// TIA Portal project "Bachelor2024" (V14)

(* hardware
DEVICE "S7-1200 station_1"  S7-1200 Station
   slot 0: "Rack_0"  S7-1200 Rack  Rack  V1.0
   slot 1: "PROFIBUS PLC"  CPU 1212C DC/DC/DC  6ES7 212-1AE40-0XB0  V4.1
   slot 101: "CM 1243-5"  CM 1243-5  6GK7 243-5DX30-0XE0  V1.3
DEVICE "GSD device_1"  GSD.Device
   slot 0: "Rack_0"  Rail
DEVICE "GSD device_2"  GSD.Device
   slot 0: "Rack_0"  Rail
DEVICE "S7-1200 station_2"  S7-1200 Station
   slot 0: "Rack_0"  S7-1200 Rack  Rack  V1.0
   slot 1: "PROFINET PLC"  CPU 1211C AC/DC/Rly  6ES7 211-1BE40-0XB0  V4.2
DEVICE "GSD device_3"  GSD.Device.PN
   slot 0: "Rack"  Rack  V1.0
   slot 0: "COUPLER (PN)"  DP/PN Coupler V1  700-158-3DP01  V 1
      slot 0: "DP/PN Coupler V1"  DP/PN Coupler V1
      slot 1: "PN-IO"  PN-IO
         slot 1: "Port 1"  Port 1
         slot 2: "Port 2"  Port 2
   slot 1: "OUT   2 Bytes_1"  OUT   2 Bytes
      slot 0: "OUT   2 Bytes"  OUT   2 Bytes
   slot 2: "IN   2 Bytes_1"  IN   2 Bytes
      slot 0: "IN   2 Bytes"  IN   2 Bytes
DEVICE "HMI"  KTP700 Basic DP
   slot 0: "KTP700 Basic DP"  KTP700 Basic DP  6AV2 123-2GA03-0AX0  14.0.1.0
   slot 1: "HMI_RT_1"  KTP700 Basic DP  6AV2 123-2GA03-0AX0  14.0.1.0
   slot 7: "HMI.MPI/DP_CP_1"  MPI/DP Interface  14.0.1.0
*)

// ===== PLC "PROFIBUS PLC"  CPU 1212C DC/DC/DC =====

VAR_GLOBAL   // PLC tag table "PUSHBUTTONS"
   "PUSHBUTTON_WHITE" AT %I0.0 : Bool;
   "PUSHBUTTON_BLUE" AT %I0.1 : Bool;
   "PUSHBUTTON_GREEN" AT %I0.2 : Bool;
   "PUSHBUTTON_ORANGE1" AT %I0.3 : Bool;
   "PUSHBUTTON_ORANGE2" AT %I0.4 : Bool;
   "PUSHBUTTON_RED" AT %I0.5 : Bool;
END_VAR

VAR_GLOBAL   // PLC tag table "FAULTS"
   "B_BREAK" AT %Q0.0 : Bool;
   "BA_BREAK" AT %Q0.1 : Bool;
   "TERMINATION_OFF" AT %Q0.2 : Bool;
   "BA_SWITCH" AT %Q0.3 : Bool;
   "NO_GROUNDING" AT %Q0.4 : Bool;
   "BA_SHORT" AT %Q0.5 : Bool;
END_VAR

VAR_GLOBAL   // PLC tag table "TESTBOARD_COUPLER"
   "TESTBOARD_INPUT1" AT %IB1 : Byte;
   "TESTBOARD_INPUT2" AT %IB2 : Byte;
   "TESTBOARD_OUTPUT1" AT %QB1 : Byte;
   "TESTBOARD_OUTPUT2" AT %QB2 : Byte;
   "COUPLER_INPUT1" AT %IB3 : Byte;
   "COUPLER_INPUT2" AT %IB4 : Byte;
   "COUPLER_OUTPUT1" AT %QB3 : Byte;
   "COUPLER_OUTPUT2" AT %QB4 : Byte;
END_VAR

// folder: System blocks/Program resources

DATA_BLOCK "IEC_Timer_0_DB"   // DB1
{ S7_Optimized_Access := 'TRUE' }
AUTHOR : Simatic
FAMILY : IEC
NAME : IEC_TMR
VERSION : 1.0
// stored: InstanceOfName IEC_TIMER
"IEC_TIMER"
BEGIN
END_DATA_BLOCK

DATA_BLOCK "IEC_Timer_0_DB_1"   // DB2
{ S7_Optimized_Access := 'TRUE' }
AUTHOR : Simatic
FAMILY : IEC
NAME : IEC_TMR
VERSION : 1.0
// stored: InstanceOfName IEC_TIMER
"IEC_TIMER"
BEGIN
END_DATA_BLOCK

DATA_BLOCK "IEC_Timer_0_DB_2"   // DB3
{ S7_Optimized_Access := 'TRUE' }
AUTHOR : Simatic
FAMILY : IEC
NAME : IEC_TMR
VERSION : 1.0
// stored: InstanceOfName IEC_TIMER
"IEC_TIMER"
BEGIN
END_DATA_BLOCK

DATA_BLOCK "IEC_Timer_0_DB_3"   // DB4
{ S7_Optimized_Access := 'TRUE' }
AUTHOR : Simatic
FAMILY : IEC
NAME : IEC_TMR
VERSION : 1.0
// stored: InstanceOfName IEC_TIMER
"IEC_TIMER"
BEGIN
END_DATA_BLOCK

DATA_BLOCK "IEC_Timer_0_DB_4"   // DB5
{ S7_Optimized_Access := 'TRUE' }
AUTHOR : Simatic
FAMILY : IEC
NAME : IEC_TMR
VERSION : 1.0
// stored: InstanceOfName IEC_TIMER
"IEC_TIMER"
BEGIN
END_DATA_BLOCK

DATA_BLOCK "IEC_Timer_0_DB_5"   // DB6
{ S7_Optimized_Access := 'TRUE' }
AUTHOR : Simatic
FAMILY : IEC
NAME : IEC_TMR
VERSION : 1.0
// stored: InstanceOfName IEC_TIMER
"IEC_TIMER"
BEGIN
END_DATA_BLOCK

// folder: (top level)

ORGANIZATION_BLOCK "Main"   // OB1, LAD, ProgramCycle
TITLE = "Main Program Sweep (Cycle)"
{ S7_Optimized_Access := 'TRUE' }
VERSION : 0.1
   VAR_INPUT
      Initial_Call : Bool;   // Initial call of this OB
      Remanence : Bool;   // =True, if remanent data are available
   END_VAR
BEGIN

REGION Network 1
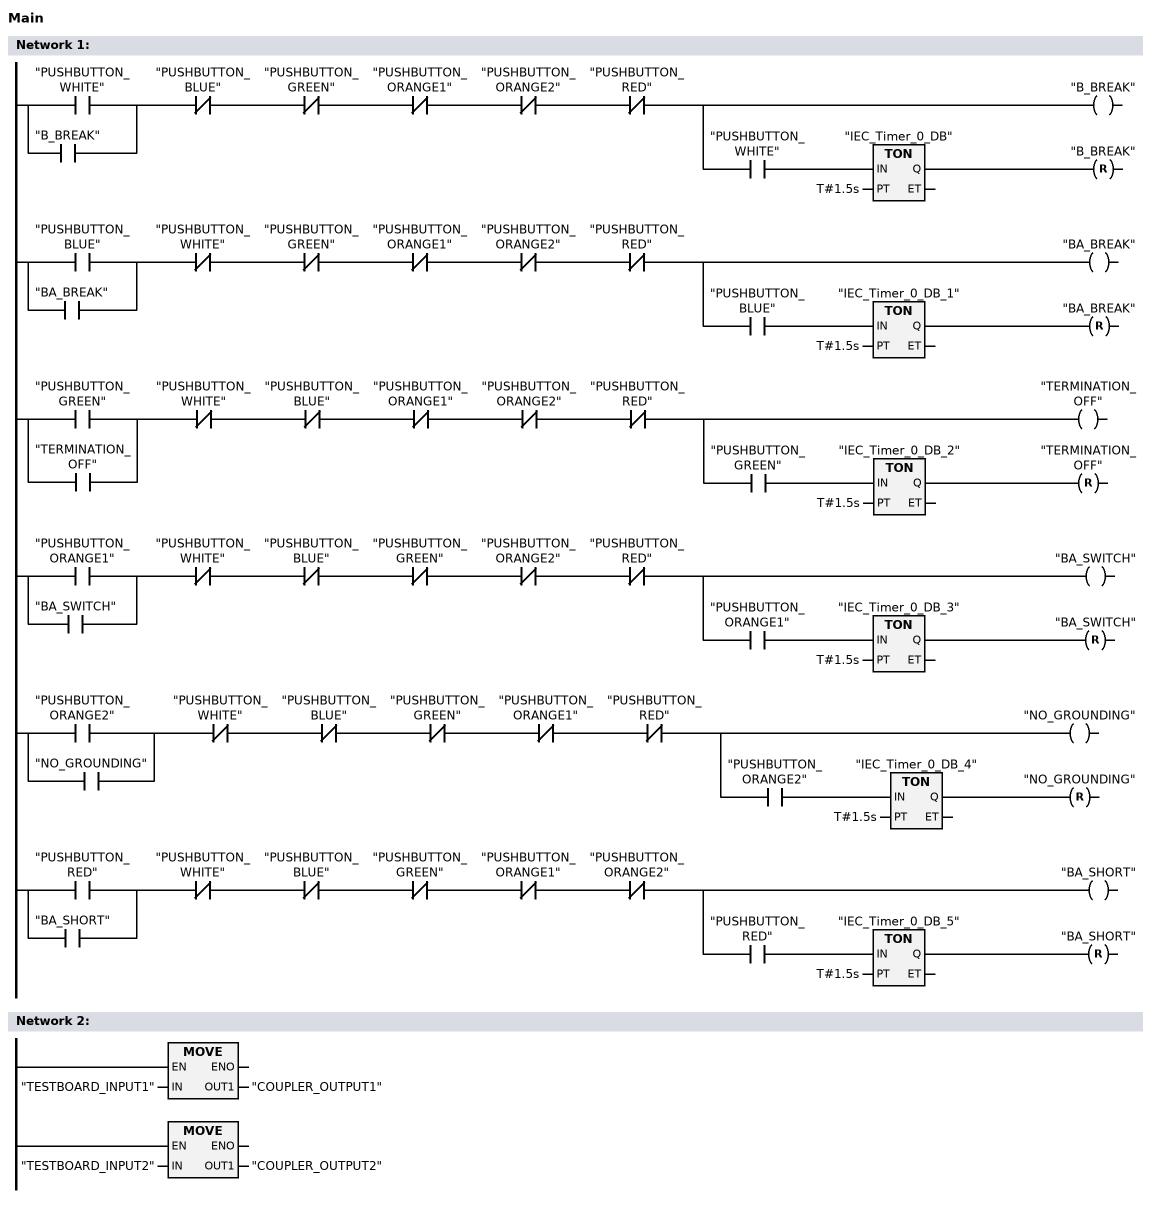
   "B_BREAK" := ("PUSHBUTTON_WHITE" OR "B_BREAK") AND NOT "PUSHBUTTON_BLUE" AND NOT "PUSHBUTTON_GREEN" AND NOT "PUSHBUTTON_ORANGE1" AND NOT "PUSHBUTTON_ORANGE2" AND NOT "PUSHBUTTON_RED";
   "IEC_Timer_0_DB".TON(IN := "B_BREAK" AND "PUSHBUTTON_WHITE", PT := T#1.5s);
   IF "IEC_Timer_0_DB".Q THEN "B_BREAK" := FALSE; END_IF;
   "BA_BREAK" := ("PUSHBUTTON_BLUE" OR "BA_BREAK") AND NOT "PUSHBUTTON_WHITE" AND NOT "PUSHBUTTON_GREEN" AND NOT "PUSHBUTTON_ORANGE1" AND NOT "PUSHBUTTON_ORANGE2" AND NOT "PUSHBUTTON_RED";
   "IEC_Timer_0_DB_1".TON(IN := "BA_BREAK" AND "PUSHBUTTON_BLUE", PT := T#1.5s);
   IF "IEC_Timer_0_DB_1".Q THEN "BA_BREAK" := FALSE; END_IF;
   "TERMINATION_OFF" := ("PUSHBUTTON_GREEN" OR "TERMINATION_OFF") AND NOT "PUSHBUTTON_WHITE" AND NOT "PUSHBUTTON_BLUE" AND NOT "PUSHBUTTON_ORANGE1" AND NOT "PUSHBUTTON_ORANGE2" AND NOT "PUSHBUTTON_RED";
   "IEC_Timer_0_DB_2".TON(IN := "TERMINATION_OFF" AND "PUSHBUTTON_GREEN", PT := T#1.5s);
   IF "IEC_Timer_0_DB_2".Q THEN "TERMINATION_OFF" := FALSE; END_IF;
   "BA_SWITCH" := ("PUSHBUTTON_ORANGE1" OR "BA_SWITCH") AND NOT "PUSHBUTTON_WHITE" AND NOT "PUSHBUTTON_BLUE" AND NOT "PUSHBUTTON_GREEN" AND NOT "PUSHBUTTON_ORANGE2" AND NOT "PUSHBUTTON_RED";
   "IEC_Timer_0_DB_3".TON(IN := "BA_SWITCH" AND "PUSHBUTTON_ORANGE1", PT := T#1.5s);
   IF "IEC_Timer_0_DB_3".Q THEN "BA_SWITCH" := FALSE; END_IF;
   "NO_GROUNDING" := ("PUSHBUTTON_ORANGE2" OR "NO_GROUNDING") AND NOT "PUSHBUTTON_WHITE" AND NOT "PUSHBUTTON_BLUE" AND NOT "PUSHBUTTON_GREEN" AND NOT "PUSHBUTTON_ORANGE1" AND NOT "PUSHBUTTON_RED";
   "IEC_Timer_0_DB_4".TON(IN := "NO_GROUNDING" AND "PUSHBUTTON_ORANGE2", PT := T#1.5s);
   IF "IEC_Timer_0_DB_4".Q THEN "NO_GROUNDING" := FALSE; END_IF;
   "BA_SHORT" := ("PUSHBUTTON_RED" OR "BA_SHORT") AND NOT "PUSHBUTTON_WHITE" AND NOT "PUSHBUTTON_BLUE" AND NOT "PUSHBUTTON_GREEN" AND NOT "PUSHBUTTON_ORANGE1" AND NOT "PUSHBUTTON_ORANGE2";
   "IEC_Timer_0_DB_5".TON(IN := "BA_SHORT" AND "PUSHBUTTON_RED", PT := T#1.5s);
   IF "IEC_Timer_0_DB_5".Q THEN "BA_SHORT" := FALSE; END_IF;
END_REGION

REGION Network 2
   RUNG wire#powerrail
      Move(in := "TESTBOARD_INPUT1", out1 => "COUPLER_OUTPUT1")
   END_RUNG
   RUNG wire#powerrail
      Move(in := "TESTBOARD_INPUT2", out1 => "COUPLER_OUTPUT2")
   END_RUNG
   // the same network as SCL:
   "COUPLER_OUTPUT1" := "TESTBOARD_INPUT1";
   "COUPLER_OUTPUT2" := "TESTBOARD_INPUT2";
END_REGION
END_ORGANIZATION_BLOCK

// ===== PLC "PROFINET PLC"  CPU 1211C AC/DC/Rly =====

VAR_GLOBAL   // PLC tag table "COUPLER_PROFINET"
   "COUPLER_INPUT1" AT %IB1 : Byte;
   "COUPLER_INPUT2" AT %IB2 : Byte;
   "COUPLER_OUTPUT1" AT %QB1 : Byte;
   "COUPLER_OUTPUT2" AT %QB2 : Byte;
END_VAR

ORGANIZATION_BLOCK "Main"   // OB1, LAD, ProgramCycle
TITLE = "Main Program Sweep (Cycle)"
{ S7_Optimized_Access := 'TRUE' }
VERSION : 0.1
   VAR_INPUT
      Initial_Call : Bool;   // Initial call of this OB
      Remanence : Bool;   // =True, if remanent data are available
   END_VAR
BEGIN

REGION Network 1
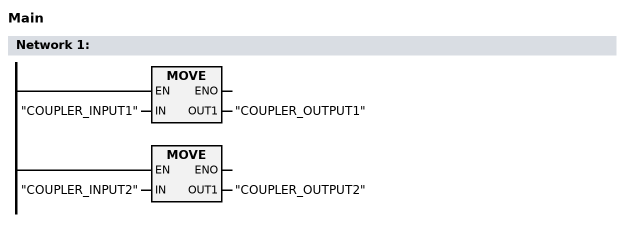
   RUNG wire#powerrail
      Move(in := "COUPLER_INPUT1", out1 => "COUPLER_OUTPUT1")
   END_RUNG
   RUNG wire#powerrail
      Move(in := "COUPLER_INPUT2", out1 => "COUPLER_OUTPUT2")
   END_RUNG
   // the same network as SCL:
   "COUPLER_OUTPUT1" := "COUPLER_INPUT1";
   "COUPLER_OUTPUT2" := "COUPLER_INPUT2";
END_REGION
END_ORGANIZATION_BLOCK

(* ===== HMI "HMI_RT_1" =====
system functions are stored by id; their names below are inferred from use
connection "HMI_Connection_1": IF1 B, SMART_S7_1200_OMS

HMI tags "Default tag table"
   "Tag_ScreenNumber" : UInt, internal

HMI tags "HMI_TAGS"
   "HMI_PUSHBUTTON_WHITE" : Bool = PLC PUSHBUTTON_WHITE AT %I0.0, 1 s
   "HMI_PUSHBUTTON_BLUE" : Bool = PLC PUSHBUTTON_BLUE AT %I0.1, 1 s
   "HMI_PUSHBUTTON_GREEN" : Bool = PLC PUSHBUTTON_GREEN AT %I0.2, 1 s
   "HMI_PUSHBUTTON_ORANGE1" : Bool = PLC PUSHBUTTON_ORANGE1 AT %I0.3, 1 s
   "HMI_PUSHBUTTON_ORANGE2" : Bool = PLC PUSHBUTTON_ORANGE2 AT %I0.4, 1 s
   "HMI_PUSHBUTTON_RED" : Bool = PLC PUSHBUTTON_RED AT %I0.5, 1 s
   "HMI_TESTBOARD_INPUT1" : Byte = PLC TESTBOARD_INPUT1 AT %IB1, 1 s
   "HMI_TESTBOARD_INPUT2" : Byte = PLC TESTBOARD_INPUT2 AT %IB2, 1 s
   "HMI_TESTBOARD_OUTPUT1" : Byte = PLC TESTBOARD_OUTPUT1 AT %QB1, 1 s
   "HMI_TESTBOARD_OUTPUT2" : Byte = PLC TESTBOARD_OUTPUT2 AT %QB2, 1 s
   "HMI_TESTBOARD_INPUT1_PN" : Byte = PLC COUPLER_INPUT1 AT %IB3, 1 s
   "HMI_TESTBOARD_INPUT2_PN" : Byte = PLC COUPLER_INPUT2 AT %IB4, 1 s

Template "Template_1" 800x480
   Button "Exit" at 714,429 size 71x50; TextOff 'Exit'; PictureOff "ExitRuntime_KTP700_Basic_DP_TR"; PictureOn "ExitRuntime_KTP700_Basic_DP_TR"
      on Release: StopRuntime(0)
   Button "Template_Button" at 614,429 size 71x50; TextOff 'Text'
   Button "Template_Button_1" at 514,429 size 71x50; TextOff 'Text'
   Button "Template_Button_2" at 414,429 size 71x50; TextOff 'Text'
   Button "Template_Button_3" at 314,429 size 71x50; TextOff 'Text'
   Button "Template_Button_4" at 214,429 size 71x50; TextOff 'Text'
   Button "Alarms" at 114,429 size 71x50; TextOff 'Alarms'; PictureOff "AlarmDisplay_KTP700_Basic_DP_TR"; PictureOn "AlarmDisplay_KTP700_Basic_DP_TR"
      on Release: function_ef3f5d25("Alarm window_Unacknowledged", -1)
   Button "Start screen" at 14,429 size 71x50; TextOff 'Start screen'; PictureOff "NavigateHome_KTP700_Basic_DP_TR"; PictureOn "NavigateHome_KTP700_Basic_DP_TR"
      on Release: ActivateScreen("Root screen", 0)
   SymbolicIOField "Symbolic_IO_Field_Screen" at 93,9 size 600x33; TextOff '0'; TextOn '1'; TextList "TextList_ScreenNames"
      ProcessValue <- "Tag_ScreenNumber"
      on Change: ActivateScreenByNumber("Tag_ScreenNumber", 0)
   DateTimeField "HmiScreenItemData" at 695,25 size 105x25
   DateTimeField "HmiScreenItemData_1" at 695,0 size 105x25
   GraphicView "Logo" at 0,0 size 91x51; Picture "Logo of HMI_1"

screen "Root screen" 800x480, template "Template_1"
   on GenerateScreen: SetTag("Tag_ScreenNumber", 1)
   Button "HmiScreenItemData" at 36,87 size 159x47; TextOff 'Screen1'; PictureOff "Navigates to Screen1 for KTP700 Basic+ DP 14.0.1.0"; PictureOn "Navigates to Screen1 for KTP700 Basic+ DP 14.0.1.0"
      on Release: ActivateScreen("Screen1", 0)
   IOField "I/O field_1" at 501,216 size 96x32; FormatPattern 999
      ProcessValue <- "HMI_TESTBOARD_INPUT1"
   IOField "I/O field_2" at 501,301 size 96x32; FormatPattern 999
      ProcessValue <- "HMI_TESTBOARD_OUTPUT1"
   TextField "Text field_1" at 437,218 size 59x23; Text 'Input1'
   TextField "Text field_2" at 425,301 size 71x23; Text 'Output1'
   TextField "Text field_3" at 525,142 size 147x23; Text 'Testboard Values'
   TextField "Text field_4" at 437,258 size 59x23; Text 'Input2'
   IOField "I/O field_3" at 501,258 size 96x32; FormatPattern 999
      ProcessValue <- "HMI_TESTBOARD_INPUT2"
   TextField "Text field_5" at 425,346 size 71x23; Text 'Output2'
   IOField "I/O field_4" at 501,342 size 96x32; FormatPattern 999
      ProcessValue <- "HMI_TESTBOARD_OUTPUT2"
   TextField "Text field_6" at 114,195 size 166x28; Text 'PUSH-BUTTONS'
   IOField "I/O field_5" at 699,216 size 96x32; FormatPattern 999
      ProcessValue <- "HMI_TESTBOARD_INPUT1_PN"
   TextField "Text field_7" at 635,218 size 59x23; Text 'Input1'
   TextField "Text field_10" at 635,258 size 59x23; Text 'Input2'
   IOField "I/O field_7" at 699,258 size 96x32; FormatPattern 999
      ProcessValue <- "HMI_TESTBOARD_INPUT2_PN"
   TextField "Text field_9" at 448,165 size 89x23; Text 'PROFIBUS'
   TextField "Text field_12" at 655,165 size 89x23; Text 'PROFINET'
   Group "Group" at 33,248 size 46x46
   Button "Button_1" at 33,248 size 46x46; TextOff '1'
      on Click: SetBit("HMI_PUSHBUTTON_WHITE")
   Button "Button_2" at 89,248 size 46x46; TextOff '2'
      on Click: SetBit("HMI_PUSHBUTTON_BLUE")
   Button "Button_3" at 145,248 size 46x46; TextOff '3'
      on Click: SetBit("HMI_PUSHBUTTON_GREEN")
   Button "Button_4" at 201,248 size 46x46; TextOff '4'
      on Click: SetBit("HMI_PUSHBUTTON_ORANGE1")
   Button "Button_5" at 257,248 size 47x46; TextOff '5'
      on Click: SetBit("HMI_PUSHBUTTON_ORANGE2")
   Button "Button_6" at 313,248 size 46x46; TextOff '6'
      on Click: SetBit("HMI_PUSHBUTTON_RED")
   GraphicView "Graphic view_2" at 468,70 size 260x48; Picture "adeptor4"

screen "Screen1" 800x480, template "Template_1"
   on GenerateScreen: SetTag("Tag_ScreenNumber", 2)
   TextField "HmiScreenItemData" at 80,225 size 640x25; Text 'Screen1'
   Button "Back" at 1,52 size 159x47; TextOff 'Back'
      on Release: ActivateScreen("Root screen", 0)
*)